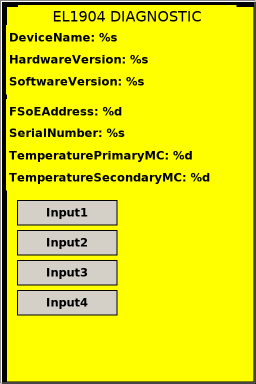
VISUALIZATION V_PH_EL1904_DIAG  // 256x384
VAR_INPUT
	stEL1904DiagnosticData		:ST_EL1904_DiagnosticData;
	
	
END_VAR
    Rectangle (2,2 256x384), colour toggle: stEL1904DiagnosticData.bGeneralError
    Rectangle (18,5 218x23), "EL1904 DIAGNOSTIC"
    Rectangle (6,25 242x25), "DeviceName: %s", text variable: stEL1904DiagnosticData.sDeviceName
    Rectangle (6,69 243x25), "SoftwareVersion: %s", text variable: stEL1904DiagnosticData.sSoftwareVersion
    Rectangle (6,47 243x25), "HardwareVersion: %s", text variable: stEL1904DiagnosticData.sHardwareVersion
    Rectangle (6,99 243x25), "FSoEAddress: %d", text variable: stEL1904DiagnosticData.dwFSoEAddress
    Rectangle (6,121 243x24), "SerialNumber: %s", text variable: stEL1904DiagnosticData.sSerialNumber
    Rectangle (6,165 243x25), "TemperatureSecondaryMC: %d", text variable: stEL1904DiagnosticData.wTemperatureSecondaryMC
    Rectangle (6,143 243x25), "TemperaturePrimaryMC: %d", text variable: stEL1904DiagnosticData.wTemperaturePrimaryMC
    RoundedRectangle (17,260 100x25), "Input3", colour toggle: stEL1904DiagnosticData.bInput3
    RoundedRectangle (17,290 100x25), "Input4", colour toggle: stEL1904DiagnosticData.bInput4
    RoundedRectangle (17,230 100x25), "Input2", colour toggle: stEL1904DiagnosticData.bInput2
    RoundedRectangle (17,200 100x25), "Input1", colour toggle: stEL1904DiagnosticData.bInput1
END_VISUALIZATION

(* stored: Version 1.1.0.1, ProductVersion 3.1.4024.4
   Visu V_PH_EL1904_DIAG: Id {831d265e-8d53-4fd3-afb0-d5d5d897b86b} *)
